{attribute 'qualified_only'}
VAR_GLOBAL
	bCoreSwagingManualMode: BOOL := FALSE;
	sAlarmMessage: STRING(50) := '';
END_VAR

(* stored: Version 1.1.0.1, ProductVersion 3.1.4024.6
   GVL GVL_HMI: Id {80a1a5a0-00a7-49c7-a368-c9a3531de34b} *)
